TYPE Type_Opt_CommOut :
STRUCT
	s_Robot		:Type_Optimization;
END_STRUCT
END_TYPE

(* stored: Version 1.1.0.1, ProductVersion 3.1.4024.3
   DUT Type_Opt_CommOut: Id {78bb90a2-5ae5-40ee-bab4-8607c26665e2} *)
